//==================================================================================================
//								RJM Maszyny sp. z o.o.
//									22.06.2022
//	Sterowanie praca maszyny   
// 	v1.0	|| TC v 3.1.4024.29		|| - pierwsza wersja
//==================================================================================================
FUNCTION_BLOCK FB_Sterowanie
VAR
	fbStart									: ITF_Przycisk;	//przycisk start
	fbStop									: ITF_Przycisk;	//przycisk stop
	fbWieza									: ITF_WiezaSygnalizacyjna;	
	bUkladSafetyOK							: BOOL;
	bWcisnietyGrzyb							: REFERENCE TO ARRAY [1..10] OF BOOL;
	iIloscGrzybowNaMaszynie					: INT := 1;
END_VAR

(* ZAŁOŻENIA
	- przelaczanie trybow
	- przelaczanie stanow 
	- przelaczanie trybow tylko w okreslonych stanach
	- reagowanie na generowanie bledow podzespolow 
	
	
*)

METHOD FB_init : BOOL
VAR_INPUT
	bInitRetains : BOOL; // if TRUE, the retain variables are initialized (warm start / cold start)
	bInCopyCode : BOOL;  // if TRUE, the instance afterwards gets moved into the copy code (online change)
	fbStart									: ITF_Przycisk;	//przycisk start
	fbStop									: ITF_Przycisk;	//przycisk stop
	fbWieza									: ITF_WiezaSygnalizacyjna;	
	bUkladSafetyOK							: BOOL;
	bWcisnietyGrzyb							: REFERENCE TO ARRAY [1..10] OF BOOL;
	iIloscGrzybowNaMaszynie					: INT;
END_VAR
THIS^.fbStart									:= fbStart;
THIS^.fbStop									:= fbStop;
THIS^.fbWieza									:= fbWieza;
THIS^.bUkladSafetyOK							:= bUkladSafetyOK;
THIS^.bWcisnietyGrzyb							:= bWcisnietyGrzyb;
THIS^.iIloscGrzybowNaMaszynie					:= iIloscGrzybowNaMaszynie;
END_METHOD

END_FUNCTION_BLOCK

(* stored: Version 1.1.0.1, ProductVersion 3.1.4024.11
   POU FB_Sterowanie: Id {13408bd3-8145-4c5f-8343-0c104b15fb7b}, SpecialFunc None
   Method FB_init: Id {d4fc2347-0397-4b16-875e-43b83cb7732a} *)
